# EPICS substitutions: eventGeneratorSup/Db/eventGenerator.substitutions
file "perFPGA.template"
{ pattern
{ P,     R,       PORT           }
  { "\$(P)", "\$(R)", "\$(PORT)" }
}

file "perBuildDate.template"
{ pattern
{       P,       R,       PORT,            NAME,        A }
  { "\$(P)", "\$(R)", "\$(PORT)",  "firmwareBuildDate", 0 }
  { "\$(P)", "\$(R)", "\$(PORT)",  "softwareBuildDate", 1 }
}

file "perSoftwareTrigger.template"
{ pattern
  {    P,      R,      PORT,   E, T,    A    }
  {"\$(P)","\$(R)","\$(PORT)", 1, 1   0x1100 }
  {"\$(P)","\$(R)","\$(PORT)", 1, 2   0x1100 }
  {"\$(P)","\$(R)","\$(PORT)", 1, 3   0x1100 }
  {"\$(P)","\$(R)","\$(PORT)", 1, 4   0x1100 }
  {"\$(P)","\$(R)","\$(PORT)", 2, 1   0x1101 }
  {"\$(P)","\$(R)","\$(PORT)", 2, 2   0x1101 }
  {"\$(P)","\$(R)","\$(PORT)", 2, 3   0x1101 }
  {"\$(P)","\$(R)","\$(PORT)", 2, 4   0x1101 }
}

file "perHardwareTrigger.template"
{ pattern
  {    P,      R,      PORT,   E, T,    A    }
  {"\$(P)","\$(R)","\$(PORT)", 1, 1   0x1200 }
  {"\$(P)","\$(R)","\$(PORT)", 1, 2   0x1201 }
  {"\$(P)","\$(R)","\$(PORT)", 1, 3   0x1202 }
  {"\$(P)","\$(R)","\$(PORT)", 1, 4   0x1203 }
  {"\$(P)","\$(R)","\$(PORT)", 1, 5   0x1204 }
  {"\$(P)","\$(R)","\$(PORT)", 1, 6   0x1205 }
  {"\$(P)","\$(R)","\$(PORT)", 1, 7   0x1206 }
  {"\$(P)","\$(R)","\$(PORT)", 1, 8   0x1207 }
  {"\$(P)","\$(R)","\$(PORT)", 2, 1   0x1210 }
  {"\$(P)","\$(R)","\$(PORT)", 2, 2   0x1211 }
  {"\$(P)","\$(R)","\$(PORT)", 2, 3   0x1212 }
  {"\$(P)","\$(R)","\$(PORT)", 2, 4   0x1213 }
  {"\$(P)","\$(R)","\$(PORT)", 2, 5   0x1214 }
  {"\$(P)","\$(R)","\$(PORT)", 2, 6   0x1215 }
  {"\$(P)","\$(R)","\$(PORT)", 2, 7   0x1216 }
  {"\$(P)","\$(R)","\$(PORT)", 2, 8   0x1217 }
}

file "perSequence.template"
{ pattern
  {    P,      R,      PORT,   E, S,  A    }
  {"\$(P)","\$(R)","\$(PORT)", 1, 0, 00 }
  {"\$(P)","\$(R)","\$(PORT)", 1, 1, 01 }
  {"\$(P)","\$(R)","\$(PORT)", 2, 0, 10 }
  {"\$(P)","\$(R)","\$(PORT)", 2, 1, 11 }
}

file "perGenerator.template"
{ pattern
  {    P,      R,      PORT,   E, I }
  {"\$(P)","\$(R)","\$(PORT)", 1, 0 }
  {"\$(P)","\$(R)","\$(PORT)", 2, 1 }
}

file "perGenericLO.template"
{ pattern
{     P     R,    PORT,             NAME,      A,             DESC }
 { \$(P),\$(R),\$(PORT),   "clrPowerup_", 0x1000, "Clear FPGA power-up status" }
 { \$(P),\$(R),\$(PORT),      "fetchTOD", 0x1002, "Resynchronize with NTP server" }
 { \$(P),\$(R),\$(PORT),"INJ:singleShot", 0x1003, "Manually trigger an injection cycle" }
 { \$(P),\$(R),\$(PORT),   "FPGA:reboot", 0x1F00, "Write 1, 100, 10000 to force reboot" }
 { \$(P),\$(R),\$(PORT),"swapoutTrigger", 0x1F02, "Trigger swapout cycle with given offset" }
 { \$(P),\$(R),\$(PORT),"MGT:Tx:realign", 0x1F03, "Write 1, 10, 100 for MGT reset/resync" }
}

file "perSysmonAI.template"
{ pattern
{     P     R,    PORT,               NAME,     A,         EGU,         ESLO,   EOFF, PREC, LOPR,  HOPR,   LOLO,    LOW,   HIGH,   HIHI,  LLSV,   LSV,   HSV,  HHSV,       DESC }
 { \$(P),\$(R),\$(PORT),       "FPGA:temp", 0x2101,"degrees C", 7.6900832e-3,-273.15,    1,    0,   100,      5,     10,     60,     68, MAJOR, MINOR, MINOR, MAJOR, "FPGA internal temperature" }
 { \$(P),\$(R),\$(PORT),   "FPGA:VccINT:V", 0x2201,        "V",  45.77636e-6,      0,    3,    0,     5,   0.90,   0.95,   1.05,   1.10, MAJOR, MINOR, MINOR, MAJOR, "FPGA VccINT voltage" }
 { \$(P),\$(R),\$(PORT),   "FPGA:VccAUX:V", 0x2102,        "V",  45.77636e-6,      0,    3,    0,     5,   1.70,   1.75,   1.85,   1.90, MAJOR, MINOR, MINOR, MAJOR, "FPGA VccAUX voltage" }
 { \$(P),\$(R),\$(PORT),  "FPGA:VccBRAM:V", 0x2202,        "V",  45.77636e-6,      0,    3,    0,     5,   0.90,   0.95,   1.05,   1.10, MAJOR, MINOR, MINOR, MAJOR, "FPGA Vcc BRAM voltage" }

 { \$(P),\$(R),\$(PORT),        "FMC1:I12", 0x2304,        "I",       5.0e-4,      0     3,    0,    20,   -0.2,   -0.1,    1.0,    1.5, MAJOR, MINOR, MINOR, MAJOR, "FMC1 supply current" }
 { \$(P),\$(R),\$(PORT),        "FMC1:V12", 0x2204,        "V",       5.0e-4,      0,    3,    0,    20,     11,  11.25,  12.75,     13, MAJOR, MINOR, MINOR, MAJOR, "FMC1 supply voltage" }
 { \$(P),\$(R),\$(PORT),        "FMC2:I12", 0x2305,        "I",       5.0e-4,      0     3,    0,    20,   -0.2,   -0.1,    1.0,    1.5, MAJOR, MINOR, MINOR, MAJOR, "FMC1 supply current" }
 { \$(P),\$(R),\$(PORT),        "FMC2:V12", 0x2205,        "V",       5.0e-4,      0,    3,    0,    20,     11,  11.25,  12.75,     13, MAJOR, MINOR, MINOR, MAJOR, "FMC1 supply voltage" }
# FIXME: Next board revision will fix the polarity of the reading
 { \$(P),\$(R),\$(PORT),      "Marble:Iin", 0x2306,        "I",-4.4117647e-4,      0     3,    0,    20,   -3.2,   -3.0,    3.0,    3.2, MAJOR, MINOR, MINOR, MAJOR, "Board supply current" }
 { \$(P),\$(R),\$(PORT),      "Marble:Vin", 0x2206,        "V",       5.0e-4,      0,    3,    0,    20,     11,  11.25,  12.75,     13, MAJOR, MINOR, MINOR, MAJOR, "Board supply voltage" }

 { \$(P),\$(R),\$(PORT),      "E1:Tx1:Vcc", 0x2107,        "V",         1e-4,      0,    3,    0,     5,   3.10,   3.20,   3.40,   3.50, MAJOR, MINOR, MINOR, MAJOR, "EVG 1 Tx 1 supply voltage" }
 { \$(P),\$(R),\$(PORT),     "E1:Tx1:temp", 0x2407,"degrees C",            1,      0,    1,    0,   100,      0,      0,     55,     65, MAJOR, MINOR, MINOR, MAJOR, "EVG 1 Tx 1 temperature" }
 { \$(P),\$(R),\$(PORT),      "E1:Rx1:Vcc", 0x2108,        "V",         1e-4,      0,    3,    0,     5,   3.10,   3.20,   3.40,   3.50, MAJOR, MINOR, MINOR, MAJOR, "EVG 1 Rx 1 supply voltage" }
 { \$(P),\$(R),\$(PORT),     "E1:Rx1:temp", 0x2408,"degrees C",            1,      0,    1,    0,   100,      0,      0,     55,     65, MAJOR, MINOR, MINOR, MAJOR, "EVG 1 Rx 1 temperature" }

 { \$(P),\$(R),\$(PORT),      "E1:Tx2:Vcc", 0x2109,        "V",         1e-4,      0,    3,    0,     5,   3.10,   3.20,   3.40,   3.50, MAJOR, MINOR, MINOR, MAJOR, "EVG 1 Tx 2 supply voltage" }
 { \$(P),\$(R),\$(PORT),     "E1:Tx2:temp", 0x2409,"degrees C",            1,      0,    1,    0,   100,      0,      0,     55,     65, MAJOR, MINOR, MINOR, MAJOR, "EVG 1 Tx 2 temperature" }
 { \$(P),\$(R),\$(PORT),      "E1:Rx2:Vcc", 0x210A,        "V",         1e-4,      0,    3,    0,     5,   3.10,   3.20,   3.40,   3.50, MAJOR, MINOR, MINOR, MAJOR, "EVG 1 Rx 2 supply voltage" }
 { \$(P),\$(R),\$(PORT),     "E1:Rx2:temp", 0x240A,"degrees C",            1,      0,    1,    0,   100,      0,      0,     55,     65, MAJOR, MINOR, MINOR, MAJOR, "EVG 1 Rx 2 temperature" }

 { \$(P),\$(R),\$(PORT),      "E1:Tx3:Vcc", 0x210B,        "V",         1e-4,      0,    3,    0,     5,   3.10,   3.20,   3.40,   3.50, MAJOR, MINOR, MINOR, MAJOR, "EVG 1 Tx 3 supply voltage" }
 { \$(P),\$(R),\$(PORT),     "E1:Tx3:temp", 0x240B,"degrees C",            1,      0,    1,    0,   100,      0,      0,     55,     65, MAJOR, MINOR, MINOR, MAJOR, "EVG 1 Tx 3 temperature" }
 { \$(P),\$(R),\$(PORT),      "E1:Rx3:Vcc", 0x210C,        "V",         1e-4,      0,    3,    0,     5,   3.10,   3.20,   3.40,   3.50, MAJOR, MINOR, MINOR, MAJOR, "EVG 1 Rx 3 supply voltage" }
 { \$(P),\$(R),\$(PORT),     "E1:Rx3:temp", 0x240C,"degrees C",            1,      0,    1,    0,   100,      0,      0,     55,     65, MAJOR, MINOR, MINOR, MAJOR, "EVG 1 Rx 3 temperature" }

 { \$(P),\$(R),\$(PORT),      "E2:Tx1:Vcc", 0x210D,        "V",         1e-4,      0,    3,    0,     5,   3.10,   3.20,   3.40,   3.50, MAJOR, MINOR, MINOR, MAJOR, "EVG 2 Tx 1 supply voltage" }
 { \$(P),\$(R),\$(PORT),     "E2:Tx1:temp", 0x240D,"degrees C",            1,      0,    1,    0,   100,      0,      0,     55,     65, MAJOR, MINOR, MINOR, MAJOR, "EVG 2 Tx 1 temperature" }
 { \$(P),\$(R),\$(PORT),      "E2:Rx1:Vcc", 0x210E,        "V",         1e-4,      0,    3,    0,     5,   3.10,   3.20,   3.40,   3.50, MAJOR, MINOR, MINOR, MAJOR, "EVG 2 Rx 1 supply voltage" }
 { \$(P),\$(R),\$(PORT),     "E2:Rx1:temp", 0x240E,"degrees C",            1,      0,    1,    0,   100,      0,      0,     55,     65, MAJOR, MINOR, MINOR, MAJOR, "EVG 2 Rx 1 temperature" }

 { \$(P),\$(R),\$(PORT),      "E2:Tx2:Vcc", 0x210F,        "V",         1e-4,      0,    3,    0,     5,   3.10,   3.20,   3.40,   3.50, MAJOR, MINOR, MINOR, MAJOR, "EVG 2 Tx 2 supply voltage" }
 { \$(P),\$(R),\$(PORT),     "E2:Tx2:temp", 0x240F,"degrees C",            1,      0,    1,    0,   100,      0,      0,     55,     65, MAJOR, MINOR, MINOR, MAJOR, "EVG 2 Tx 2 temperature" }
 { \$(P),\$(R),\$(PORT),      "E2:Rx2:Vcc", 0x2110,        "V",         1e-4,      0,    3,    0,     5,   3.10,   3.20,   3.40,   3.50, MAJOR, MINOR, MINOR, MAJOR, "EVG 2 Rx 2 supply voltage" }
 { \$(P),\$(R),\$(PORT),     "E2:Rx2:temp", 0x2410,"degrees C",            1,      0,    1,    0,   100,      0,      0,     55,     65, MAJOR, MINOR, MINOR, MAJOR, "EVG 2 Rx 2 temperature" }

 { \$(P),\$(R),\$(PORT),      "E2:Tx3:Vcc", 0x2111,        "V",         1e-4,      0,    3,    0,     5,   3.10,   3.20,   3.40,   3.50, MAJOR, MINOR, MINOR, MAJOR, "EVG 2 Tx 3 supply voltage" }
 { \$(P),\$(R),\$(PORT),     "E2:Tx3:temp", 0x2411,"degrees C",            1,      0,    1,    0,   100,      0,      0,     55,     65, MAJOR, MINOR, MINOR, MAJOR, "EVG 2 Tx 3 temperature" }
 { \$(P),\$(R),\$(PORT),      "E2:Rx3:Vcc", 0x2112,        "V",         1e-4,      0,    3,    0,     5,   3.10,   3.20,   3.40,   3.50, MAJOR, MINOR, MINOR, MAJOR, "EVG 2 Rx 3 supply voltage" }
 { \$(P),\$(R),\$(PORT),     "E2:Rx3:temp", 0x2412,"degrees C",            1,      0,    1,    0,   100,      0,      0,     55,     65, MAJOR, MINOR, MINOR, MAJOR, "EVG 2 Rx 3 temperature" }

 { \$(P),\$(R),\$(PORT),        "U28:temp", 0x2319,"degrees C",          0.5,      0,    1,    0,   100,      2,      5,     55,     65, MAJOR, MINOR, MINOR, MAJOR, "Marble U28 temperature" }
 { \$(P),\$(R),\$(PORT),        "U29:temp", 0x2419,"degrees C",          0.5,      0,    1,    0,   100,      2,      5,     55,     65, MAJOR, MINOR, MINOR, MAJOR, "Marble U29 temperature" }

 { \$(P),\$(R),\$(PORT),    "E1:refJitter", 0x221A,       "ps",       13.167,      0,    1,    0,  1000,     -1,     -1,    180,    250, MAJOR, MINOR, MINOR, MAJOR, "EVG 1 refClk sampled by EVG 2 refClk" }
 { \$(P),\$(R),\$(PORT),     "E1:txJitter", 0x221B,       "ps",       13.167,      0,    1,    0,  1000,     -1,     -1,    180,    250, MAJOR, MINOR, MINOR, MAJOR, "EVG 1 txClk sampled by EVG 2 refClk" }
 { \$(P),\$(R),\$(PORT),    "E1:frequency", 0x201C,      "MHz",         1e-6,      0,    6,    0,   200,    123,    124,    126,    127, MAJOR, MINOR, MINOR, MAJOR, "EVG 1 reference clock rate" }
 { \$(P),\$(R),\$(PORT),    "E2:refJitter", 0x221D,       "ps",       13.167,      0,    1,    0,  1000,     -1,     -1,    180,    250, MAJOR, MINOR, MINOR, MAJOR, "EVG 2 refClk sampled by EVG 1 refClk" }
 { \$(P),\$(R),\$(PORT),     "E2:txJitter", 0x221E,       "ps",       13.167,      0,    1,    0,  1000,     -1,     -1,    180,    250, MAJOR, MINOR, MINOR, MAJOR, "EVG 2 txClk sampled by EVG 1 refClk" }
 { \$(P),\$(R),\$(PORT),    "E2:frequency", 0x201F,      "MHz",         1e-6,      0,    6,    0,   200,    123,    124,    126,    127, MAJOR, MINOR, MINOR, MAJOR, "EVG 2 reference clock rate" }
}

file "perSysmonLI.template"
{ pattern
{     P     R,    PORT,          NAME,             A,      EGU,               DESC }
 { \$(P),\$(R),\$(PORT),        "Marble:PIO_", 0x2003,       "", "Marble port expanders" }

 { \$(P),\$(R),\$(PORT)     "E1:Rx1:enabled",  0x2113,       "", "Enabled receivers (bitmap)" }
 { \$(P),\$(R),\$(PORT)     "E1:Rx1:lowPower", 0x2213,       "", "Receivers with low power (bitmap)" }
 { \$(P),\$(R),\$(PORT)     "E1:Rx2:enabled",  0x2114,       "", "Enabled receivers (bitmap)" }
 { \$(P),\$(R),\$(PORT)     "E1:Rx2:lowPower", 0x2214,       "", "Receivers with low power (bitmap)" }
 { \$(P),\$(R),\$(PORT)     "E1:Rx3:enabled",  0x2115,       "", "Enabled receivers (bitmap)" }
 { \$(P),\$(R),\$(PORT)     "E1:Rx3:lowPower", 0x2215,       "", "Receivers with low power (bitmap)" }
 { \$(P),\$(R),\$(PORT)     "E2:Rx1:enabled",  0x2116,       "", "Enabled receivers (bitmap)" }
 { \$(P),\$(R),\$(PORT)     "E2:Rx1:lowPower", 0x2216,       "", "Receivers with low power (bitmap)" }
 { \$(P),\$(R),\$(PORT)     "E2:Rx2:enabled",  0x2117,       "", "Enabled receivers (bitmap)" }
 { \$(P),\$(R),\$(PORT)     "E2:Rx2:lowPower", 0x2217,       "", "Receivers with low power (bitmap)" }
 { \$(P),\$(R),\$(PORT)     "E2:Rx3:enabled",  0x2118,       "", "Enabled receivers (bitmap)" }
 { \$(P),\$(R),\$(PORT)     "E2:Rx3:lowPower", 0x2218,       "", "Receivers with low power (bitmap)" }

 { \$(P),\$(R),\$(PORT),        "E1:refCoinc", 0x211A, "counts", "EVG 1 refClk sampled by EVG 2 refClk" }
 { \$(P),\$(R),\$(PORT),         "E1:txCoinc", 0x211B, "counts", "EVG1 txClk sampled by EVG 2 refClk" }
 { \$(P),\$(R),\$(PORT),        "E2:refCoinc", 0x211D, "counts", "EVG2 refClk sampled by EVG 1 refClk" }
 { \$(P),\$(R),\$(PORT),         "E2:txCoinc", 0x211E, "counts", "EVG2 txClk sampled by EVG 1 refClk" }
 { \$(P),\$(R),\$(PORT),    "INJ:injCycleCSR", 0x2021,       "", "Injection sequence CSR" }
 { \$(P),\$(R),\$(PORT),         "TOD:Status", 0x2022,       "", "TOD valid 1:Seconds 0:PPS" }
 { \$(P),\$(R),\$(PORT),    "E1:EVIOstatus_",  0x2123,       "", "EVG 1 raw status" }
 { \$(P),\$(R),\$(PORT),    "E2:EVIOstatus_",  0x2223,       "", "EVG 2 raw status" }
 { \$(P),\$(R),\$(PORT),    "swapoutstatus_",  0x2024,       "", "Swapout control status register" }
 { \$(P),\$(R),\$(PORT),     "E1:MGTstatus_",  0x2027,       "", "EVG 1 raw MGT status" }
 { \$(P),\$(R),\$(PORT),     "E2:MGTstatus_",  0x2028,       "", "EVG 2 raw MGT status" }
 { \$(P),\$(R),\$(PORT), "INJ:AlignstatusSlow_", 0x2029,     "", "Injection align status" }
 { \$(P),\$(R),\$(PORT), "swapoutAlignstatusSlow_", 0x202A,  "", "Swapout align status" }
}

file "perSysmonBI.template"
{ pattern
{     P     R,    PORT,          NAME,          A,        ZNAM,      ONAM,       ZSV,        OSV,         DESC }
 { \$(P),\$(R),\$(PORT), "EVG:aligned",    0x2120,"Misaligned", "Aligned",   "MAJOR", "NO_ALARM", "Are generators aligned" }
}

file "perSysmonFan.template"
{ pattern
{     P     R,    PORT,  N,     A, }
 { \$(P),\$(R),\$(PORT), 1, 0x2325 }
 { \$(P),\$(R),\$(PORT), 2, 0x2425 }
 { \$(P),\$(R),\$(PORT), 3, 0x2326 }
 { \$(P),\$(R),\$(PORT), 4, 0x2426 }
}
